PROGRAM Echange_OPCUA
VAR
	Ton_NT_GetTime:Ton;
	fbGetTime:NT_GetTime;
	
	{attribute 'OPC.UA.DA' := '1'}
	stTIMESTR: Tc2_Utilities.TIMESTRUCT;
END_VAR

fbGetTime(
	NETID:= '', 
	START:= Ton_NT_GetTime.Q, 
	TMOUT:= DEFAULT_ADS_TIMEOUT, 
	BUSY=> , 
	ERR=> , 
	ERRID=> , 
	TIMESTR=> stTIMESTR);
	
	
Ton_NT_GetTime(IN:= NOT fbGetTime.BUSY , PT:=T#500MS , Q=> , ET=> );

END_PROGRAM

(* stored: Version 1.1.0.1, ProductVersion 3.1.4026.18
   POU Echange_OPCUA: Id {2ca0bbd9-d188-4c20-ba0b-1c64a6c14ad1}, SpecialFunc None *)
